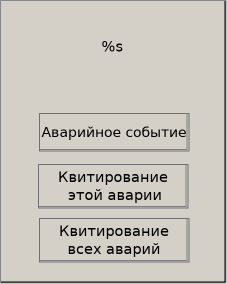
VISUALIZATION tAlarm  // 227x284
VAR_IN_OUT
	alarm: FB_Alarm;
END_VAR
    Rectangle (0,0 225x282), "%s", text variable: alarm.AlarmInfo.Description, colour toggle: Tc3_BAR_Common.LibAlarm.Blink and alarm.isActive
    Button (39,113 150x38), "Аварийное событие"
        toggle alarm.AlarmEvent
    Button (38,164 150x44), "Квитирование этой аварии"
        tap alarm.bQuitAlarm
    Button (39,218 150x44), "Квитирование всех аварий"
        tap Tc3_BAR_Common.LibAlarm.bLocalQuitAllAlarms
END_VISUALIZATION

(* stored: Version 1.1.0.1, ProductVersion 3.1.4024.2
   Visu tAlarm: Id {4b04ca6c-075b-485f-9fe2-d2a59d780c8c} *)
